// TwinCAT 3 PLC project Bangsarebuilding
// ProgramVersion: 3.1.4023.0
// libraries:
//   Tc2_EnOcean, * (Beckhoff Automation GmbH)
//   Tc2_Standard, * (Beckhoff Automation GmbH)
//   Tc2_System, * (Beckhoff Automation GmbH)
//   Tc2_Utilities, * (Beckhoff Automation GmbH)
//   Tc3_IotBase, * (Beckhoff Automation GmbH)
//   Tc3_Module, * (Beckhoff Automation GmbH)
// project tree:
//   %40Main/ MAIN.TcPOU (not stored)
//   DUTs/ ST_FrameData.TcDUT
//   / GlobalTextList.TcGTLO, PlcTask.TcTTO, Visualization Manager.TcVMO (not stored)
//   GVLs/ GVLKL3403.TcGVL, GVLmqtt.TcGVL, GVL_Enocean.TcGVL, GVL_HouseControl.TcGVL, GVL_IO_Enocean.TcGVL, GVL_RTClock.TcGVL
//   POUs/AverageLog/ FB_LoggAverage.TcPOU, NewAverage.TcPOU
//   POUs/CurrentMeassuring/ CurrentMeassuring.TcPOU, KL3403_FB.TcPOU
//   POUs/DataExchange/ DataExchange.TcPOU, F_Checksum.TcPOU
//   POUs/Enocean/ Control.TcPOU, Enocean_program.TcPOU
//   POUs/HouseControlProgram/ HouseControl.TcPOU
//   POUs/MQTT/ FB_MyMqtt.TcPOU, PrgMqttCom.TcPOU
//   POUs/RTClock/ RTClock.TcPOU
//   VISUs/VisuEnocean/ TC_VISU.TcVIS
// real-time tasks:
//   TASK PlcTask: cycle T#10ms, priority 20, ADS port 350
// I/O:
//   DEVICE Device 1 (CX-BK)
//     Box 1 (CX-BK)
// variable links:
//   Bangsarebuilding/Bangsarebuilding Instance <-> Device 1 (CX-BK)/Box 1 (CX-BK)
//     PlcTask Inputs/.DATAIN/nData <-> Term 10 (KL6021-0023)/Channel 1/Data In 0
//     PlcTask Inputs/.DATAIN/nData @bit 8 <-> Term 10 (KL6021-0023)/Channel 1/Data In 1
//     PlcTask Inputs/.DATAIN/nData @bit 80 <-> Term 10 (KL6021-0023)/Channel 1/Data In 10
//     PlcTask Inputs/.DATAIN/nData @bit 16 <-> Term 10 (KL6021-0023)/Channel 1/Data In 2
//     PlcTask Inputs/.DATAIN/nData @bit 24 <-> Term 10 (KL6021-0023)/Channel 1/Data In 3
//     PlcTask Inputs/.DATAIN/nData @bit 32 <-> Term 10 (KL6021-0023)/Channel 1/Data In 4
//     PlcTask Inputs/.DATAIN/nData @bit 40 <-> Term 10 (KL6021-0023)/Channel 1/Data In 5
//     PlcTask Inputs/.DATAIN/nData @bit 48 <-> Term 10 (KL6021-0023)/Channel 1/Data In 6
//     PlcTask Inputs/.DATAIN/nData @bit 56 <-> Term 10 (KL6021-0023)/Channel 1/Data In 7
//     PlcTask Inputs/.DATAIN/nData @bit 64 <-> Term 10 (KL6021-0023)/Channel 1/Data In 8
//     PlcTask Inputs/.DATAIN/nData @bit 72 <-> Term 10 (KL6021-0023)/Channel 1/Data In 9
//     PlcTask Inputs/.DATAIN/nStatus <-> Term 10 (KL6021-0023)/Channel 1/nStatus
//     PlcTask Inputs/.KL3403_DataIn_3 <-> Term 14 (KL3403)/Channel 1/.KL3403_DataIn_3
//     PlcTask Inputs/.KL3403_State_1 <-> Term 14 (KL3403)/Channel 1/.KL3403_State_1
//     PlcTask Inputs/.PT100_BathRoom <-> Term 13 (KL3204)/Channel 2/.PT100_BathRoom
//     PlcTask Inputs/.PT100_CX1000 <-> Term 13 (KL3204)/Channel 3/.PT100_CX1000
//     PlcTask Inputs/.PT100_Outside <-> Term 13 (KL3204)/Channel 1/.PT100_Outside
//     PlcTask Inputs/.Term3204_4_Data_In <-> Term 13 (KL3204)/Channel 4/.Term3204_4_Data_In
//     PlcTask Outputs/.AeLight <-> Term 7 (KL2012)/Channel 2/.AeLight
//     PlcTask Outputs/.AirBedroom <-> Term 3 (KL2641)/Channel 1/.AirBedroom
//     PlcTask Outputs/.AirBjorn <-> Term 2 (KL2641)/Channel 1/.AirBjorn
//     PlcTask Outputs/.BedRoomLight <-> Term 6 (KL2012)/Channel 1/.BedRoomLight
//     PlcTask Outputs/.BjornLight <-> Term 9 (KL2012)/Channel 1/.BjornLight
//     PlcTask Outputs/.DATAOUT/nCtrl <-> Term 10 (KL6021-0023)/Channel 1/nCtrl
//     PlcTask Outputs/.EntranceLight <-> Term 5 (KL2012)/Channel 2/.EntranceLight
//     PlcTask Outputs/.KL3403_Ctrl_1 <-> Term 14 (KL3403)/Channel 1/.KL3403_Ctrl_1
//     PlcTask Outputs/.KL3403_DataOut_3 <-> Term 14 (KL3403)/Channel 1/Data Out
//     PlcTask Outputs/.Livingroom <-> Term 6 (KL2012)/Channel 2/.Livingroom
//     PlcTask Outputs/.ReceptionLight <-> Term 5 (KL2012)/Channel 1/Output
//     PlcTask Outputs/.Spare <-> Term 8 (KL2012)/Channel 1/.Spare
//     PlcTask Outputs/.StairLight <-> Term 9 (KL2012)/Channel 2/.StairLight
//     PlcTask Outputs/.ToiletLight <-> Term 8 (KL2012)/Channel 2/.ToiletLight
//     PlcTask Outputs/.WalkingClosett <-> Term 7 (KL2012)/Channel 1/.WalkingClosett

CONFIGURATION Bangsarebuilding
    RESOURCE PLC ON TwinCAT3
        TASK PlcTask(INTERVAL := T#10ms, PRIORITY := 20);
        PROGRAM MAIN WITH PlcTask : MAIN;
    END_RESOURCE
END_CONFIGURATION

// ---- DUTs/ST_FrameData.TcDUT
(* 8 byte aligned structure, byte size := 152 byte *)
TYPE ST_FrameData :
STRUCT
    nFrameSize: DWORD;(*Frame byte size, member byte size := 4 byte*)
    nTxFrames : DWORD;(*Tx frame number, member byte size := 4 byte*)
    nRxFrames : DWORD;(*Rx frame number, member byte size := 4 byte*)
    nCounter  : DWORD;(*Number value, member byte size := 4 byte*)
    fU        : REAL;(*Floating point number, member byte size := 4 byte*)
    fV        : REAL;(*Floating point number, member byte size := 4 byte*)
    fW        : REAL;(*Floating point number, member byte size := 4 byte*)
    aFloats   : ARRAY[0..9] OF REAL;(* Array of floating point numbers, array byte size := 40 byte*)
    sMsg      : STRING;(*String variable, member byte size := 81 byte incl. String null delimiter*)
    bEnable   : BOOL;(*Boolean flag, member byte size := 1 byte*)
    nRsv0     : BYTE;(*Reserved byte to meet the 8 byte alignment, member byte size := 1 byte*)
    nCRC      : BYTE;(*CRC checksum byte, member byte size := 1 byte*)
END_STRUCT
END_TYPE

// ---- GVLs/GVLKL3403.TcGVL
{attribute 'Tc2GvlVarNames'}
VAR_GLOBAL
	KL3403_Ctrl_1 		AT %Q*: USINT;
	KL3403_State_1		AT %I* 	:USINT;
	KL3403_DataOut_1	 AT %Q*: INT;
	KL3403_DataIn_1	 	AT %I*	: INT;
	KL3403_Ctrl_2 		AT %Q*	: USINT;
	KL3403_State_2		AT %I* 	:USINT;
	KL3403_DataOut_2	 AT %Q*	: INT;
	KL3403_DataIn_2 		AT %I*	: INT;
	KL3403_Ctrl_3 		AT %Q*	: USINT;
	KL3403_State_3		AT %I* 	:USINT;
	KL3403_DataOut_3	 AT %Q*	: INT;
	KL3403_DataIn_3 		AT %I*	: INT;

	intOutputStatus: INT;
END_VAR

// ---- GVLs/GVLmqtt.TcGVL
{attribute 'qualified_only'}
VAR_GLOBAL

END_VAR

// ---- GVLs/GVL_Enocean.TcGVL
{attribute 'Tc2GvlVarNames'}
VAR_GLOBAL
	SummaryWordForBoolenM6 : WORD;
	OutsideTemp		: INT; 
	STM1556 :INT;

	BjornTemp 			: INT;
	OfficeTemp		 	: INT;
	BedRoomTemp 		: INT;
(* Check if enocean varible has hanged*)
	EnableForAllPTM100: BOOL := TRUE;
	CheckIfEnoceanSwitchIsPressed: DWORD;
	SRW01State: BOOL;
(*Viewer Variables*)
	EnOceanEasyClick  : BYTE; (* Status bSwitches in EnOceanEasyClick*)
	EnOceanPTM100SWbjorn :BYTE;(* Status bSwitches in EnOceanPTM100SW*)
	EnOceanPTM100SWentrance : BYTE;(* Status bSwitches in EnOceanPTM100SWentrance*)

	SRO4PeEnOceanRotarySwitch: E_EnOceanRotarySwitch;
	SRO4Psetpoint: INT;
	SRO4bPresentSwitch: BOOL;
	SRO4PbLearnSwitch: BOOL;

	SRO4P_2eEnOceanRotarySwitch: E_EnOceanRotarySwitch;
	SRO4P_2setpoint: INT;
	SRO4_2bPresentSwitch: BOOL;
	SRO4_2PbLearnSwitch: BOOL;

	SRO4P_3eEnOceanRotarySwitch: E_EnOceanRotarySwitch;
	SRO4P_3setpoint: INT;
	SRO4_3bPresentSwitch: BOOL;
	SRO4P_3bLearnSwitch: BOOL;

	SRO4PeEnOceanRotarySwitch4: E_EnOceanRotarySwitch;
	SRO4Psetpoint4: INT;
	SRO4bPresentSwitch4: BOOL;
	SRO4PbLearnSwitch4: BOOL;

(*Timers*)
	TurnLightsOffTimer: TON;
	ShutAllOff: TON;


(* Variables*)

	bLearnSTM250: BOOL;
	EnoceanResieved: ST_EnOceanReceivedData;
	EnOceanPTM100SSpareAndToilet: BYTE;
	SPir360data: ARRAY [0..3] OF BYTE;


	SRO4b3PresentSwitch: BOOL;
	SRO4P3bLearnSwitch: BOOL;
	ShutAllOff_ElapsedTime: STRING(80);
	
//	PlaceHolder_IfLightsAreON		AT %QX13.7	: BOOL;		


//	Control_ifLightsAreON 			AT %QW12: WORD;
(*	OutputControl_ifLightsAreON 				AT %QW128: WORD; (Summary word for Boolean below
	InputControl_ifLightsAreON					AT %IW132: WORD; (Summary word for Boolean below *)
END_VAR

// ---- GVLs/GVL_HouseControl.TcGVL
{attribute 'qualified_only'}
VAR_GLOBAL
//ShutAllOff(); //Maybee for later use
//ShutAllOff_ElapsedTime :=DELETE( LEFT(TIME_TO_STRING(ShutAllOff.PT-ShutAllOff.ET),5),3,0);
END_VAR

// ---- GVLs/GVL_IO_Enocean.TcGVL
{attribute 'Tc2GvlVarNames'}
VAR_GLOBAL
	DATAIN 		AT %I*: ST_EnOceanInData;
	DATAOUT 	AT %Q*: ST_EnOceanOutData;
	SpotLight		AT %Q*:	BOOL;
	ReceptionLight	AT %Q*:	BOOL;
	EntranceLight	AT %Q*:	BOOL;
	BedRoomLight	AT %Q*:	BOOL;
	Livingroom		AT %Q*:	BOOL;
	WalkingClosett	AT %Q*:	BOOL;
	AeLight			AT %Q*:	BOOL;
	BjornLight		AT %Q*:	BOOL;
	StairLight		AT %Q*:	BOOL;
	ToiletLight		AT %Q*:	BOOL;
	Spare			AT %Q*:	BOOL;
	AirBjorn 		AT %Q*: BOOL ;		
	AirBedroom 		AT %Q*: BOOL;
	TotalCurrent :	 	 INT;
	PT100_Outside		AT %I*: INT;
//	Term3403_Ctrl_1		AT %Q*: USINT;
//	Term3403_DataOut_1	AT %Q*: INT;
	PT100_BathRoom 		AT %I*: INT;
//	Term3403_Ctrl_2 		AT %Q*: USINT;
//	Term3403_DataOut_2	AT %Q*: INT;
	PT100_CX1000 		AT %I*: INT;
//	Term3403_Ctrl_3 		AT %Q*: USINT;
//	Term3403_DataOut_3	AT %Q*: INT;
//	Term3204_1_State		AT %I*:	USINT;
//	Term3204_1_Data_In	AT %I*:	INT; (*Outside*)
//	Term3204_1_Ctrl		AT %Q*:	USINT;
//	Term3204_1_Data_Out	AT %Q*:	INT;
//	Term3204_2_State		AT %IB4:USINT;
//	Term3204_2_Data_In	AT %I*:	INT;
//	Term3204_2_Ctrl		AT %Q*:	USINT;
//	Term3204_2_Data_Out	AT %Q*:	INT;
//	Term3204_3_State		AT %I*:	USINT;
//	Term3204_3_Data_In	AT %I*:	INT;
//	Term3204_3_Ctrl		AT %Q*:	USINT;
//	Term3204_3_Data_Out	AT %Q*:	INT;
//	Term3204_4_State		AT %I*:	USINT;
	Term3204_4_Data_In	AT %I*:	INT;
//	Term3204_4_Ctrl		AT %Q*:	USINT;
//	Term3204_4_Data_Out	AT %Q*:	INT;
END_VAR

// ---- GVLs/GVL_RTClock.TcGVL
{attribute 'Tc2GvlVarNames'}
VAR_GLOBAL
	stTime: TIMESTRUCT;
	PCTime: STRING;
	bRTCValid: BOOL;
	bOldWeekend: BOOL;
	OldWorkinghour: BOOL;
	OldDay: DWORD;
	OldHour: DWORD;
	OldMinute: DWORD;
//	OldSecond: DWORD;
	OldMounth: WORD;
	ChangeOfMounth: BOOL;
(*Change Variabler togels if Var has changed*)
	ChangeWeekend: BOOL;
	ChangeOfweek :BOOL;
	ChangeWorkingHour: BOOL;
	ChangeOfDay: BOOL;
	bHourChanged: BOOL;
	bMinuteChanged : BOOL;
//	bSecondCanged: BOOL;
(* Detect status*)
	bWeekend: BOOL;
	WorkingHour: BOOL;
	OldYear: WORD;
END_VAR

// ---- POUs/AverageLog/FB_LoggAverage.TcPOU
FUNCTION_BLOCK FB_LoggAverage
VAR_INPUT
	usTimeBase: USINT;(* In time i.e 60  for seconds and minutes or 24 for Hour *)
	wTIMSTR : WORD;
	rLoggdata : LREAL;
END_VAR
VAR_OUTPUT
	rAverage :LREAL ;
	arrIntern: ARRAY[0..59] OF LREAL;
END_VAR
VAR
	i: USINT;
	rMinuteAverage:  LREAL;
	//y: INT := 100;
	//: BOOL;
	//bTest: BOOL;
	usZero: USINT;
	bTimeChanged: BOOL;
	OldTimestring: WORD;	
	//arrIntern: ARRAY[0..59] OF LREAL;
END_VAR

//VAR_INPUT //old ver
//	usTimeBase: USINT;(* In time i.e 60  for seconds and minutes or 24 for Hour *)
//	wTIMSTR : WORD;
//	rLoggdata : LREAL;
//END_VAR
//VAR_OUTPUT
//	rAverage :LREAL ;
//	arrIntern : ARRAY[0..59] OF LREAL;
//END_VAR
//VAR
//	i: USINT;
//	rMinuteAverage:  LREAL;
//	y: INT := 100;
//	bFillArr: BOOL;
//	bTest: BOOL;
//	usZero: USINT;
//	bTimeChanged: BOOL;
//END_VAR

IF wTIMSTR = OldTimestring THEN
;
ELSE
bTimeChanged:= TRUE;
END_IF
OldTimestring:=wTIMSTR;
IF bTimeChanged THEN
rMinuteAverage :=0;
 arrIntern[wTIMSTR] := rLoggdata;
	IF wTIMSTR= usTimeBase -1   THEN
	usZero := usTimeBase;
		FOR i := 0 TO usTimeBase -1  DO
			IF arrIntern[i] = 0 THEN
			usZero := usZero - 1;
			END_IF
		rMinuteAverage := arrIntern[i]+ rMinuteAverage;
arrIntern[i] := 0;

 			IF i = usTimeBase -1 THEN
				IF usZero = 0 THEN
				RETURN ;
				END_IF
	 		rAverage := rMinuteAverage / (usZero ) ;
			bTimeChanged := FALSE ;
			END_IF
		END_FOR
	END_IF
END_IF

END_FUNCTION_BLOCK

// ---- POUs/AverageLog/NewAverage.TcPOU
PROGRAM NewAverage
VAR
	rAverageMin: LREAL;
	rAverageHour: LREAL;
	rAverageDay : LREAL;
	rLoggData: LREAL ;
	FB_LoggAverageMonth: FB_LoggAverage;
	FB_LoggAverageDays:  FB_LoggAverage;
	FB_LoggAverageHours: FB_LoggAverage;
	FB_LoggAverageMinutes: FB_LoggAverage;
	FB_LoggAverageSeconds: FB_LoggAverage;
(*	arrZeros : ARRAY[0..9 ]  OF sDataLogg; *)

	rTestData: REAL;
	rAverageMonth: LREAL;
	rAverageYear: LREAL;
END_VAR


rLoggData := .TotalCurrent; //Test
FB_LoggAverageSeconds(
	usTimeBase:=60 ,
	wTIMSTR := GVL_RTClock.stTime.wSecond, (* Array index *)
	rLoggData:= rLoggData ,							(**)
	rAverage=> rAverageMin);

FB_LoggAverageMinutes(
	usTimeBase:=60 ,
	wTIMSTR := GVL_RTClock.stTIME. wMinute, (* Array index *)
	rLoggData:= rAverageMin ,							(**)
	rAverage=> rAverageHour );

FB_LoggAverageHours(
	usTimeBase:=24 ,
	wTIMSTR := GVL_RTClock.stTIME. wHour  , (* Array index *)
	rLoggData:= rAverageHour ,
	rAverage=> rAverageDay) ;

FB_LoggAverageDays( 
	usTimeBase:= 31,
	wTIMSTR := GVL_RTClock.stTime.wDay, (* Array index *)
	rLoggData:= rAverageDay ,
	rAverage =>rAverageMonth);

FB_LoggAverageMonth( 
	usTimeBase:= 31,
	wTIMSTR := GVL_RTClock.stTime.wMonth, (* Array index *)
	rLoggData:= rAverageMonth ,
	rAverage =>rAverageYear);

END_PROGRAM

// ---- POUs/CurrentMeassuring/CurrentMeassuring.TcPOU
PROGRAM CurrentMeassuring
VAR
	bEnable: BOOL := TRUE;
	arrPowerMeasure1: ARRAY [0..11] OF INT;
	arrPowerMeasure2 : ARRAY [0..11] OF INT;
	arrPowerMeasure3 : ARRAY [0..11] OF INT;
	fb_Ch1: KL3403_FB;
(*	fb_Ch2: KL3403_FB;
	fb_Ch3: KL3403_FB;*)
	intOldHour: INT;
	arrLoggHour: ARRAY [0..1,0..23] OF REAL;
	intOldDay: INT;
	arrDataYesterday: ARRAY [0..1,0..23] OF REAL;
	realCurrentRMS: REAL;
	realVoltageRMS: REAL;
	realEff_Power: REAL;
	realPF: REAL;
	realPeakCurrent: REAL;
	realPeakVoltage: REAL;
	realPeakPower: REAL;
	realHz: REAL;
	realMinCurrent: REAL;
	realMinVoltage: REAL;
END_VAR
VAR_INPUT
	intState: USINT;
END_VAR

(*
fb_Ch1(
	bEnable:= TRUE,
	usintState:= KL3403_State_1,
	intDataIN:=KL3403_DataIn_1 ,
	usintCTRL=>KL3403_Ctrl_1 ,
	arrPowerMeasure => arrPowerMeasure1,
	realCurrentRMS=> intCurrentLamp1,
	realVoltageRMS=>intVoltage1


fb_Ch2(
	bEnable:= TRUE,
	usintState:= KL3403_State_2,
	intDataIN:=KL3403_DataIn_2 ,
	usintCTRL=>KL3403_Ctrl_2 ,
	arrPowerMeasure => arrPowerMeasure2,
	realCurrentRMS=> intCurrentLamp2,
	realVoltageRMS=>intVoltage2
 );
 *)
fb_Ch1(
	bEnable:= TRUE,
	usintState:= KL3403_State_3,
	intDataIN:=KL3403_DataIn_3 ,
	usintCTRL=>KL3403_Ctrl_3 ,
	arrPowerMeasure => arrPowerMeasure3,
//	realCurrentRMS=>intCurrentSolar ,
//	realVoltageRMS=>intVoltage3
 );

arrPowerMeasure1[0];
arrPowerMeasure1[1];
.TotalCurrent := KL3403_DataIn_3;

fb_Ch1(
	bEnable:= bEnable,
	usintState:= KL3403_State_3,
	intDataIN:= KL3403_DataIn_3,
	usintCTRL=>KL3403_Ctrl_3 ,
	arrPowerMeasure => arrPowerMeasure2,
	realCurrentRMS=> realCurrentRMS, 
	realVoltageRMS=>realVoltageRMS ,
	realEff_Power=>realEff_Power , 
	realPF=>realPF , 
	realEnergyConsumtion=> , 
	realPeakCurrent=>realPeakCurrent ,
	realPeakVoltage=> realPeakVoltage,
	realPeakPower=> realPeakPower, 
	realHz=>realHz , 
	realMinCurrent=> realMinCurrent, 
	realMinVoltage=> realMinVoltage, 
	realMinPower=> realMinVoltage );

END_PROGRAM

// ---- POUs/CurrentMeassuring/KL3403_FB.TcPOU
FUNCTION_BLOCK KL3403_FB
VAR
	TP1: TP;
	TP2: TP;
	R_TRIG1: R_TRIG;

	INDEX: BYTE;
	CurrentRMS: REAL;
	VoltageRMS: REAL;
	EffectivePower: REAL;
	PowerFactor: REAL;
	EnergyConsuntion: REAL;
	PeakCurrent: REAL;
	PeakVoltage: REAL;
	PeakPower: REAL;
	Frequency: REAL;
	MinimumCurrent: REAL;
	MinimumVoltage: REAL;
	MinimumPower: REAL;
END_VAR
VAR_INPUT
	bEnable: BOOL;
	usintState : INT;
	intDataIN: INT;
END_VAR
VAR_OUTPUT
	usintCTRL: USINT;
	arrPowerMeasure: ARRAY [0..11] OF INT;
	realCurrentRMS: REAL;
	realVoltageRMS: REAL;
	realEff_Power: REAL;
	realPF: REAL;
	realEnergyConsumtion: REAL;
	realPeakCurrent: REAL;
	realPeakVoltage: REAL;
	realPeakPower: REAL;
	realHz: REAL;
	realMinCurrent: REAL;
	realMinVoltage: REAL;
	realMinPower: REAL;
END_VAR

(* Update Value form KL3403*)

usintCTRL := index ;
IF usintState.0 = usintCTRL.0 THEN
arrPowerMeasure[index] := intDataIN ;
index := index +1;
END_IF
IF index >11 THEN Index := 0 ; END_IF

(*Transfer data*)


(*Show in Function Block Output*)
realCurrentRMS :=INT_TO_REAL (arrPowerMeasure[0]);
realVoltageRMS := INT_TO_REAL (arrPowerMeasure[1])/10.0;
realEff_Power := INT_TO_REAL( arrPowerMeasure[2]);
realPF := INT_TO_REAL (arrPowerMeasure[3] ) ;
realEnergyConsumtion := INT_TO_REAL (arrPowerMeasure[4] ) ;
realPeakCurrent := INT_TO_REAL (arrPowerMeasure[4]) ;
realPeakVoltage := INT_TO_REAL (arrPowerMeasure[4])/10.0;
realPeakPower := INT_TO_REAL (arrPowerMeasure[4]) ;
realHz :=INT_TO_REAL (arrPowerMeasure[4])/10.0;
realMinCurrent := INT_TO_REAL( arrPowerMeasure[4]);
realMinVoltage := INT_TO_REAL (arrPowerMeasure[4] )/ 10.0;
realMinPower := INT_TO_REAL (arrPowerMeasure[4]);

END_FUNCTION_BLOCK

// ---- POUs/DataExchange/DataExchange.TcPOU
PROGRAM DataExchange
VAR
    bWrite        : BOOL;(* Rising edge at this variable writes data to the BC/BX (Bus Terminal Controller) *)
    bRead         : BOOL;(* Rising edge at this variable reads data from BC/BX (Bus Terminal Controller) *)
    stTxFrame     : ST_FrameData; (* Data transported from PC/CX (x86) to BC/BX (Bus Terminal Contoroller) *)
    stRxFrame     : ST_FrameData; (* Data transported from BC/BX (Bus Terminal Controller) to PC/CX (x86) *)
    fbWrite       : ADSWRITE :=  ( NETID := '172.16.5.128.1.1', PORT := 800, IDXGRP := 16#4020, IDXOFFS := 500, TMOUT := DEFAULT_ADS_TIMEOUT );
    fbRead        : ADSREAD :=  ( NETID := '172.16.5.128.1.1', PORT := 800, IDXGRP := 16#4020, IDXOFFS := 0, TMOUT := DEFAULT_ADS_TIMEOUT );
    (* Temporary used variables *)
    stTxToBC      : ST_FrameData;
    stRxFromBC    : ST_FrameData;
    i             : INT;
    nTxState      : UDINT;
    nRxState      : UDINT;
    nTxErrors     : UDINT;
    nRxErrors     : UDINT;
END_VAR

(*##########################################################################################*)
CASE nTxState OF
    0:
        IF bWrite THEN(* Write BC/BX data *)
            bWrite := FALSE;

            (* Prepare/modify tx data *)
            stTxFrame.nFrameSize    := SIZEOF( stTxFrame );(* Set frame byte size *)
            stTxFrame.nTxFrames    := stTxFrame.nTxFrames + 1;(* Increment the send frame number *)
            stTxFrame.nRxFrames     := stRxFrame.nTxFrames;(* Report the received frame number *)
            stTxFrame.bEnable    := NOT stTxFrame.bEnable;(* Toggle bool flag *)
            stTxFrame.nCounter     := stTxFrame.nCounter + 1;(* Increment counter value *)
            stTxFrame.sMsg         := CONCAT( 'Message from PC/CX, counter: ', DWORD_TO_STRING( stTxFrame.nCounter ) );(* Create some string message *)
            stTxFrame.fU            := stTxFrame.fU + 1.2;(* Modify some floating point values *)
            stTxFrame.fV            := stTxFrame.fV + 3.4;
            stTxFrame.fW            := stTxFrame.fW + 5.6;
            FOR i:= 0 TO 9 DO
                stTxFrame.aFloats[i] := stTxFrame.aFloats[i] + i;
            END_FOR
            stTxFrame.nCRC         := 0;

            (* Create temporary copy of tx data *)
            stTxToBC := stTxFrame;

            (* Swap REAL variables to BC/BX (Bus Terminal Controller) format *)
            F_SwapRealEx( stTxToBC .fU );
            F_SwapRealEx( stTxToBC .fV );
            F_SwapRealEx( stTxToBC .fW );
            FOR i:= 0 TO 9 DO
                F_SwapRealEx( stTxToBC .aFloats[i] );
            END_FOR
    
            (* Create CRC check number *)
            stTxToBC .nCRC     := F_CheckSum( ADR( stTxToBC ), SIZEOF( stTxToBC ) - 1 );
    
            (* Send *)
            fbWrite( WRITE := FALSE );
            fbWrite( LEN := SIZEOF( stTxToBC ), SRCADDR := ADR( stTxToBC ), WRITE := TRUE );
            nTxState := 1;
        END_IF

    1:(* Wait until ads write command not busy *)
        fbWrite( WRITE := FALSE );
        IF NOT fbWrite.BUSY THEN
            IF NOT fbWrite.ERR THEN
                nTxState := 0;
            ELSE(* Ads error *)
                nTxState := 100;
            END_IF
        END_IF

    100: (* TODO: Error state, add error handling *)
        nTxErrors := nTxErrors + 1;
        nTxState := 0;

END_CASE

(*##########################################################################################*)
CASE nRxState OF
    0:
        IF bRead THEN(* Read BC/BX data *)
            bRead := FALSE;

            fbRead( READ := FALSE );
            fbRead( LEN := SIZEOF( stRxFromBC ), DESTADDR := ADR( stRxFromBC ), READ := TRUE );
            nRxState := 1;
        END_IF

    1:(* Wait until ads read command not busy *)
        fbRead( READ := FALSE );
        IF NOT fbRead.BUSY THEN
            IF NOT fbRead.ERR THEN
                (* Perform simple frame length check *)
                IF stRxFromBC.nFrameSize = SIZEOF( stRxFromBC ) THEN (* Check frame length *)
                    (* Perform simple CRC check *)
                    IF stRxFromBC.nCRC = F_CheckSum( ADR( stRxFromBC ), SIZEOF( stRxFromBC ) - 1 ) THEN

                        (* Swap REAL variables to PC/CX (x86) format *)
                        F_SwapRealEx( stRxFromBC.fU );
                        F_SwapRealEx( stRxFromBC.fV );
                        F_SwapRealEx( stRxFromBC.fW );
                        FOR i:= 0 TO 9 DO
                            F_SwapRealEx( stRxFromBC.aFloats[i] );
                        END_FOR

                        stRxFrame := stRxFromBC;
                        nRxState     := 0;

                    ELSE(* => Checksum error *)
                        nRxState := 100;
                    END_IF
                ELSE(* => Invalid frame length *)
                    nRxState := 100;
                END_IF
            ELSE(* => Ads error *)
                nRxState := 100;
            END_IF
        END_IF

    100: (* TODO: Error state, add error handling *)
        nRxErrors := nRxErrors + 1;
        nRxState := 0;

END_CASE

END_PROGRAM

// ---- POUs/DataExchange/F_Checksum.TcPOU
FUNCTION F_Checksum : BYTE
VAR_INPUT
	pBuffer 		: POINTER TO BYTE;
	cbBuffer 	: UDINT;
END_VAR
VAR
	i			: UDINT;
END_VAR

IF ( pBuffer = 0 ) OR ( cbBuffer = 0 ) THEN
	F_CheckSum := 0;
	RETURN;
END_IF

FOR i:= 1 TO cbBuffer DO
	F_CheckSum := F_CheckSum + pBuffer^;
	pBuffer := pBuffer + 1;
END_FOR

END_FUNCTION

// ---- POUs/Enocean/Control.TcPOU
PROGRAM Control
VAR
	rtrigStairs: R_TRIG;
	rtrigBjorn: R_TRIG;
	rtrigBalcony: R_TRIG;
	rtrigWindow: R_TRIG;
	rtrigToilet: R_TRIG;
	rtrigBedroom: R_TRIG;
	rtrigEntrance: R_TRIG;
	rtrigSofa: R_TRIG;
	rtrigSpotlight: R_TRIG;
	rtrigReception: R_TRIG;
	rtrigEntrance2: R_TRIG;
	rtrigSofa2: R_TRIG;
	rtrigSpotlight2: R_TRIG;
	rtrigReception2: R_TRIG;
	rtrigPreparationToLeave: R_TRIG;
	Delay: TIME := T#10S;
	OffTimerPTM100SWbjorn: TON;
	OffTimerPTM100SWentrance:TON;
	OffTimerEasyClick:TON;
	OffTimerSpareAndToilet: TON;
	OldSummaryWordForBoolenM6: WORD;
	VBchange: BOOL;
	TON_InputHanged: TON;
	TimerFoorAirBedroom: TON;
	WorkingHourTest: BOOL;
	rtrig4: R_TRIG;
	rtrig5: R_TRIG;
	rtrig1: R_TRIG;
	rtrig0: R_TRIG;
	A: UINT;
	bTest: BOOL;
END_VAR



Control.EasyfitBjorn();(* Action uses data from Switch at Room Bjorn*)
Control.EasyFitSpareAndToiletUppstairs();(* Action uses data from Switch at Spareroom and Toilet uppstairs*)
Control.EasyfitEntrance(); (* Action uses data from Switch at entrance door*)

ACTION EasyfitBjorn:
(* EasyfitBjornEasyfitEntrance has 4 buttons, controling 4 lamps press a button is on and if same button is prssed more than 1sec light goes off
Data is evalueted in MAIN.EntrancewitchControl.EnOceanPTM100SWbjorn, i.e. .bSw0 to bSw3 are set when corresponding switch is pressed *)

rtrigStairs(CLK:=Enocean_program.fb_PTM100SWbjorn1159899.bSwitches[4] );
rtrigBjorn(CLK := Enocean_program.fb_PTM100SWbjorn1159899.bSwitches[5]);
rtrigBalcony(CLK := Enocean_program.fb_PTM100SWbjorn1159899.bSwitches[1]);
rtrigWindow(CLK := Enocean_program.fb_PTM100SWbjorn1159899.bSwitches[0]);

IF rtrigStairs.Q THEN
StairLight := NOT StairLight;
END_IF
IF rtrigBalcony.Q THEN
	Livingroom:= NOT Livingroom ;
END_IF
IF rtrigBjorn.Q THEN
	BjornLight :=NOT BjornLight;
END_IF
IF rtrigWindow.Q THEN
	BedRoomLight := NOT BedRoomLight;
END_IF
END_ACTION

ACTION EasyfitEntrance:
(* EasyfitEntrance has 4 buttons, controling 4 lamps. 2 Switches doing the same jobb are used *)

rtrigEntrance(CLK:= Enocean_program.fb_PTM100SWentrance1119127.bSwitches[5]  );
rtrigSofa(CLK:=  Enocean_program.fb_PTM100SWentrance1119127.bSwitches[1] );
rtrigSpotlight(CLK:= Enocean_program.fb_PTM100SWentrance1119127.bSwitches[4]   );
rtrigReception(CLK:= Enocean_program.fb_PTM100SWentrance1119127.bSwitches[0]  );
(*
rtrigEntrance2(CLK:= Enocean_program.fb_PTM100SWentrance1119127.bSwitches[5]  );
rtrigSofa2(CLK:=  Enocean_program.fb_PTM100SWentrance1119127.bSwitches[1] );
rtrigSpotligh2t(CLK:= Enocean_program.fb_PTM100SWentrance1119127.bSwitches[4]   );
rtrigReception2(CLK:= Enocean_program.fb_PTM100SWentrance1119127.bSwitches[0]  );
*)


(*Turn On and Off  Light at Entrance*)

IF rtrigEntrance.Q  THEN(* Upper left switch *)
	ReceptionLight := NOT ReceptionLight;
END_IF
IF rtrigSofa.Q  THEN(*Lower Left SW*)
	AeLight := NOT AeLight;
	(*IF NOT DayTime THEN	Stairs :=TRUE; END_IF*)
END_IF

IF rtrigSpotlight.Q THEN (* Upper right switch *)
	SpotLight := NOT SpotLight;
END_IF
IF rtrigReception.Q THEN(*Lower Left SW*)
	ReceptionLight := NOT ReceptionLight;
END_IF

(*
IF rtrigEntrance2.Q  THEN(* Upper left switch *)
	Entrance := NOT Entrance;
END_IF
IF rtrigSofa2.Q  THEN(*Lower Left SW*)
	Sofa := NOT Sofa;
	IF NOT WorkingHour THEN	Stairs :=TRUE; END_IF
END_IF

IF rtrigSpotlight2.Q THEN (* Upper right switch *)
	Spotlight := NOT Spotlight;
END_IF
IF rtrigReception2.Q THEN(*Lower Left SW*)
	Reception := NOT Reception;
END_IF
*)
END_ACTION

ACTION EasyFitSpareAndToiletUppstairs:
(* EasyFitSpareAndToiletUppstairs has 2buttons, controling 2 lamps press a button is on and if same button is prssed more than 1sec light goes off
Data is evalueted in MAIN.EntrancewitchControl.EasyFitSpareAndToiletUppstairs, i.e. .bSw0 to bSw3 are set when corresponding switch is pressed *)
rtrigToilet (CLK:= Enocean_program.fb_PTM100SWSpareAndToilet1075788.bSwitches[5] , Q=> );
rtrigBedroom(CLK:= Enocean_program.fb_PTM100SWSpareAndToilet1075788.bSwitches[1]  , Q=> );
IF rtrigToilet.Q  THEN
	ToiletLight:=NOT ToiletLight;
END_IF
IF rtrigBedroom.Q THEN
	BedRoomLight := NOT  BedRoomLight;
END_IF
END_ACTION

END_PROGRAM

// ---- POUs/Enocean/Enocean_program.TcPOU
PROGRAM Enocean_program (* Evaluates in _RECIVER if an Enocean signal is activated
							the other fb:s controls variables  depending on Enoceandata recieved.*)
VAR_INPUT
END_VAR
VAR
	FB_EnOceanReceive1: FB_EnOceanReceive;
	fb_BeckhoffSooftSW4294378625	:FB_EnOceanPTM100;
	fb_PTM100SWentrance1119127		: FB_EnOceanPTM100;
	fb_PTM100SWbjorn1159899			: FB_EnOceanPTM100;
	fb_PTM100SWSpareAndToilet1075788: FB_EnOceanPTM100;
	FB_EnOceanSTM100				: FB_EnOceanSTM100;
	FB_EnOceanSTM1556				: FB_EnOceanSTM100;
	FB_EnOceanSTM100_2				: FB_EnOceanSTM100;
	FB_EnOceanSTM100_3				: FB_EnOceanSTM100;
	FB_EnOceanSTM100_4				: FB_EnOceanSTM100;
	FB_EnOceanSTM250				: FB_EnOceanSTM250;
	FB_EnOceanSTM100PIR360			: FB_EnOceanSTM100Generic;
	bSwitches:ARRAY[0..7] OF BOOL ;
	bError: BOOL;
	nErrorId: UDINT;
	PresentTransmiterId: UDINT;
	FB_EnOceanReceive2: FB_EnOceanReceive;
	ui1556: INT;
	ui1936: INT;
	ui58058: INT;
	ui58059: INT;
	ui58398: INT;
END_VAR

(*1138914  Evaluates in _RECIVER if an Enocean signal  is activated, the other fb:s sets a variables  depending on Enoceandata recieved.*)
FB_EnOceanReceive1(
	bEnable:= TRUE, 
	bError=> , 
	nErrorId=> , 
	stEnOceanReceivedData=> EnoceanResieved, 
	stEnOceanInData:= DATAIN , 
	stEnOceanOutData:= DATAOUT);
//FB_EnOceanReceive1				(
//								bEnable:=TRUE ,
//								stEnOceanInData:=DATAIN ,
//								stEnOceanOutData:=DATAOUT ,	
//								bError=> ,	
//								nErrorId=> ,	
//								stEnOceanReceivedData=>EnoceanResieved );
								
fb_PTM100SWentrance1119127	(bEnable:= EnableForAllPTM100,	tWatchdog:=,	nTransmitterId:=1119127 ,	stEnOceanReceivedData:= FB_EnOceanReceive1.stEnOceanReceivedData,
										bSwitches=>,	bError=> ,	nErrorId=> );
fb_PTM100SWbjorn1159899		(	bEnable:= EnableForAllPTM100,	tWatchdog:=,	nTransmitterId:= 1159899,	stEnOceanReceivedData:= FB_EnOceanReceive1.stEnOceanReceivedData,
										bSwitches=>,	bError=> ,	nErrorId=> );
fb_PTM100SWSpareAndToilet1075788(	bEnable:= EnableForAllPTM100,	tWatchdog:=,	nTransmitterId:= 1075788,	stEnOceanReceivedData:= FB_EnOceanReceive1.stEnOceanReceivedData,
										bSwitches=>,	bError=> ,	nErrorId=> );
fb_BeckhoffSooftSW4294378625 (bEnable:= EnableForAllPTM100,
							    tWatchdog:=,	nTransmitterId:= 1406393,
								stEnOceanReceivedData:= FB_EnOceanReceive1.stEnOceanReceivedData,
								bSwitches=>bSwitches,
								bError=>bError ,
								nErrorId=>nErrorId );

FB_EnOceanSTM100					(bEnable:=TRUE ,	tWatchdog:=T#30m ,	nTransmitterId:=58398 ,	stEnOceanReceivedData:=FB_EnOceanReceive1.stEnOceanReceivedData ,
										 eEnOceanRotarySwitch=>SRO4PeEnOceanRotarySwitch  ,	nSetpoint=>SRO4Psetpoint ,	nTemperature=> ,	bPresentSwitch=>SRO4bPresentSwitch ,
										bLearnSwitch=>SRO4PbLearnSwitch ,bError=> ,	nErrorId=> );
FB_EnOceanSTM1556					(bEnable:=TRUE ,	tWatchdog:=T#30M ,	nTransmitterId:=1556 ,	stEnOceanReceivedData:=FB_EnOceanReceive1.stEnOceanReceivedData ,
										 eEnOceanRotarySwitch=>SRO4PeEnOceanRotarySwitch  ,	nSetpoint=>SRO4Psetpoint ,	nTemperature=> ,	bPresentSwitch=>SRO4bPresentSwitch ,
										bLearnSwitch=>SRO4PbLearnSwitch ,bError=> ,	nErrorId=> );										
FB_EnOceanSTM100_2			(	bEnable:=TRUE ,	tWatchdog:=T#30m ,	nTransmitterId:=58058 ,	stEnOceanReceivedData:=FB_EnOceanReceive1.stEnOceanReceivedData ,
										eEnOceanRotarySwitch=>SRO4P_2eEnOceanRotarySwitch  ,	nSetpoint=>SRO4P_2setpoint ,	nTemperature=> ,	bPresentSwitch=>SRO4_2bPresentSwitch ,
										bLearnSwitch=>SRO4_2PbLearnSwitch ,	bError=> ,	nErrorId=> );
FB_EnOceanSTM100_3			(	bEnable:=TRUE ,	tWatchdog:=T#30m ,	nTransmitterId:=58059 ,	stEnOceanReceivedData:=FB_EnOceanReceive1.stEnOceanReceivedData ,
										eEnOceanRotarySwitch=>SRO4PeEnOceanRotarySwitch  ,	nSetpoint=>SRO4P_3setpoint ,	nTemperature=> ,	bPresentSwitch=>SRO4_3bPresentSwitch ,
										bLearnSwitch=>SRO4P_3bLearnSwitch ,	bError=> ,	nErrorId=> );
FB_EnOceanSTM100_4			(	bEnable:=TRUE ,	tWatchdog:=T#30m ,	nTransmitterId:=1936 ,	stEnOceanReceivedData:=FB_EnOceanReceive1.stEnOceanReceivedData ,
										eEnOceanRotarySwitch=>SRO4PeEnOceanRotarySwitch4  ,	nSetpoint=>SRO4Psetpoint4 ,	nTemperature=> ,	bPresentSwitch=>SRO4bPresentSwitch4 ,
										bLearnSwitch=>SRO4PbLearnSwitch4 ,	bError=> ,	nErrorId=> );

FB_EnOceanSTM100PIR360		(	bEnable:=TRUE ,	tWatchdog:=T#30m ,	nTransmitterId:=41490 ,	stEnOceanReceivedData:=FB_EnOceanReceive1.stEnOceanReceivedData ,
										nDataBytes=>SPir360data ,	bError=> ,	nErrorId=> );
FB_EnOceanSTM250				(	bEnable:=TRUE ,	tWatchdog:= ,	nTransmitterId:=25391 ,	stEnOceanReceivedData:=FB_EnOceanReceive1.stEnOceanReceivedData,
										bState=>SRW01State ,	bLearn=> bLearnSTM250,	bError=> , 	nErrorId=> );

(* Temperature is present in 1/10 grad i.e 312 means 31.2 grad*)
PresentTransmiterId:=EnoceanResieved.nTransmitterId;
 CASE PresentTransmiterId OF
1556: ui1556 := ui1556 + 1;	 
1936: ui1936 := ui1936 + 1;
58058: ui58058 := ui58058 + 1;
58059: ui58059 := ui58059 + 1;
58398:	ui58398 := ui58398 + 1; 
 END_CASE
OutsideTemp  :=FB_EnOceanSTM100.nTemperature;
OfficeTemp :=FB_EnOceanSTM100_2.nTemperature ;
STM1556 := FB_EnOceanSTM1556.nTemperature ;
BedRoomTemp :=FB_EnOceanSTM100_3.nTemperature ;
BjornTemp:=FB_EnOceanSTM100_4.nTemperature;


(* the array bSwitches is really 8 BYTE using only 1 bit as Boolean.
Below they are converted to bit in 1 WORD. evaluated in CheckIfHanged*) 
EnOceanEasyClick.0 :=FB_BeckhoffSooftSW4294378625.bSwitches[0];
EnOceanEasyClick.1 :=FB_BeckhoffSooftSW4294378625.bSwitches[1];
EnOceanEasyClick.4 :=FB_BeckhoffSooftSW4294378625.bSwitches[4];
EnOceanEasyClick.5 :=FB_BeckhoffSooftSW4294378625.bSwitches[5];

EnOceanPTM100SWbjorn.0 :=fb_PTM100SWbjorn1159899.bSwitches[0];
EnOceanPTM100SWbjorn.1 :=fb_PTM100SWbjorn1159899.bSwitches[1];
EnOceanPTM100SWbjorn.4 :=fb_PTM100SWbjorn1159899.bSwitches[4];
EnOceanPTM100SWbjorn.5 :=fb_PTM100SWbjorn1159899.bSwitches[5];

EnOceanPTM100SWentrance.0 :=fb_PTM100SWentrance1119127.bSwitches[0];
EnOceanPTM100SWentrance.1 :=fb_PTM100SWentrance1119127.bSwitches[1];
EnOceanPTM100SWentrance.4 :=fb_PTM100SWentrance1119127.bSwitches[4];
EnOceanPTM100SWentrance.5 :=fb_PTM100SWentrance1119127.bSwitches[5];

EnOceanPTM100SSpareAndToilet.1 :=fb_PTM100SWSpareAndToilet1075788.bSwitches[1];
EnOceanPTM100SSpareAndToilet.5 :=fb_PTM100SWSpareAndToilet1075788.bSwitches[5];

(*
Not used in PTM Switch with 2 channels
EnOceanPTM100SSpareAndToilet.0 :=fb_PTM100SWSpareAndToilet1075788.bSwitches[0];
EnOceanPTM100SSpareAndToilet.2 :=fb_PTM100SWSpareAndToilet1075788.bSwitches[2];
EnOceanPTM100SSpareAndToilet.3 :=fb_PTM100SWSpareAndToilet1075788.bSwitches[3];
EnOceanPTM100SSpareAndToilet.4 :=fb_PTM100SWSpareAndToilet1075788.bSwitches[4];
EnOceanPTM100SSpareAndToilet.6 :=fb_PTM100SWSpareAndToilet1075788.bSwitches[6];
EnOceanPTM100SSpareAndToilet.7 :=fb_PTM100SWSpareAndToilet1075788.bSwitches[7];
*)

END_PROGRAM

// ---- POUs/HouseControlProgram/HouseControl.TcPOU
PROGRAM HouseControl
VAR

END_VAR


IF stTime.wHour = 18 AND stTime.wMinute =1 THEN
StairLight := TRUE; //Cant be shut off for 1 minute 
ELSIF stTime.wHour = 23 AND stTime.wMinute =59 THEN
StairLight := TRUE; //Cant be shut off for 1 minute 	
END_IF

END_PROGRAM

// ---- POUs/MQTT/FB_MyMqtt.TcPOU
{attribute 'c++_compatible'}
FUNCTION_BLOCK FB_MyMqtt EXTENDS FB_IotMqttClient
VAR_INPUT
END_VAR
VAR_OUTPUT
END_VAR

VAR
	(* received message *)
	{attribute 'TcEncoding':='UTF-8'}
	sTopicRcv : STRING(255);
	{attribute 'TcEncoding':='UTF-8'}
	sPayloadRcv : STRING(255);
	A: BOOL;
	nVar: INT;
END_VAR

{attribute 'c++_compatible'}
{attribute 'pack_mode' := '4'}
{attribute 'show'}
{attribute 'minimal_input_size' := '4'}
METHOD OnMqttMessage : HRESULT
VAR_IN_OUT CONSTANT
	topic	: STRING;
END_VAR
VAR_INPUT
	payload	: PVOID;
	length	: UDINT;
	qos	: TcIotMqttQos;
	repeated	: BOOL;
END_VAR

VAR
	sRecived: STRING(255);
Test :int ;
END_VAR
SUPER^.nMessagesRcv := SUPER^.nMessagesRcv + 1;

STRNCPY( ADR(sTopicRcv), ADR(topic), SIZEOF(sTopicRcv) );
MEMCPY( ADR(sPayloadRcv), payload, MIN(length, DINT_TO_UDINT(SIZEOF(sPayloadRcv))) );
sTopicRcv;
sPayloadRcv;
nVar := STRING_TO_INT(sPayloadRcv);
IF sTopicRcv = 'BangsareLights' THEN
      CASE nVar OF 
		  0: ;
		  1:  SpotLight := NOT SpotLight;
		  2:  ReceptionLight := NOT ReceptionLight ;
		  3:  EntranceLight := NOT EntranceLight;
		  4:  BedRoomLight := NOT BedRoomLight;
		  5:  Livingroom := NOT Livingroom;
		  6:  WalkingClosett := NOT WalkingClosett;
		  7:  BjornLight := FALSE;
		  8:  BjornLight := TRUE;
		  9:  StairLight := FALSE;
		  10: StairLight := TRUE;
		  11: Spare := NOT Spare;
	  END_CASE
	  	Test :=Test +1;
	END_IF
	sPayloadRcv:='0';
OnMqttMessage := S_OK;
END_METHOD

END_FUNCTION_BLOCK

// ---- POUs/MQTT/PrgMqttCom.TcPOU
PROGRAM PrgMqttCom
VAR
	fbMqttClient : FB_MyMqtt;
	bSetParameter : BOOL := TRUE;
	bConnect : BOOL := TRUE;
	
	(* published message *)
	sTopicPub : STRING(255) := 'MyTopic';
	sPayloadPub : STRING(255);
	i: UDINT;
	fbTimer : TON := (PT:=T#1S);
	
	bSubscribed : BOOL;
	sTopicSub : STRING(255) := 'MyTopic';
	
	hrErrorOccurred : HRESULT; // contains the latest occurred error
	fbTimerET: TIME;
	bFbTimer: BOOL;
	Value: UDINT;
END_VAR

IF bSetParameter THEN
	bSetParameter := FALSE;
	fbMqttClient.sHostName:= 'SERVICE';
	fbMqttClient.nHostPort:= 1883;
	fbMqttClient.sClientId:= 'IotMqttSample'; 
	fbMqttClient.sTopicPrefix:= ''; 
//	fbMqttClient.nKeepAlive:= 60; 
//	fbMqttClient.sUserName:= ;
//	fbMqttClient.sUserPassword:= ; 
//	fbMqttClient.stTLS:= ;
 	fbMqttClient.stWill.sTopic := 'LASTWILL';
//	fbMqttClient.stWill.pPayload:= 'IotMqttSample';
	fbMqttClient.stWill.nPayloadSize := Value;
END_IF

fbMqttClient.Execute(bConnect);
IF fbMqttClient.bError THEN
	// add your error logging here
	hrErrorOccurred := fbMqttClient.hrErrorCode;
END_IF
//Add Subscribe here
IF fbMqttClient.bConnected THEN
	IF NOT bSubscribed THEN
		bSubscribed := fbMqttClient.Subscribe(sTopic:=sTopicSub, eQoS:=TcIotMqttQos.AtMostOnceDelivery);
		bSubscribed := fbMqttClient.Subscribe(sTopic:='motorCurrent', eQoS:=TcIotMqttQos.AtMostOnceDelivery);
		bSubscribed := fbMqttClient.Subscribe(sTopic:='motorTemp', eQoS:=TcIotMqttQos.AtMostOnceDelivery);
		bSubscribed := fbMqttClient.Subscribe(sTopic:='motorVoltage', eQoS:=TcIotMqttQos.AtMostOnceDelivery);
		bSubscribed := fbMqttClient.Subscribe(sTopic:='BangsareLights', eQoS:=TcIotMqttQos.AtMostOnceDelivery);
		IF fbMqttClient.bError THEN
			// add your error logging here
			hrErrorOccurred := fbMqttClient.hrErrorCode;
		END_IF
	END_IF
	//Add Publish here
	fbTimer(IN:=bFbTimer , PT:=T#10S , Q=> , ET=>fbTimerET );
	IF fbTimer.Q THEN // publish new payload every second // Changed to minute
		fbTimer(IN:=FALSE);
		i := i + 1;
		sPayloadPub := CONCAT('MyMessage', TO_STRING(i));
		fbMqttClient.Publish(	sTopic:= sTopicPub, 
								pPayload:= ADR(sPayloadPub), nPayloadSize:= LEN2(ADR(sPayloadPub))+1, 
								eQoS:= TcIotMqttQos.AtMostOnceDelivery, bRetain:= FALSE, bQueue:= FALSE );
		IF fbMqttClient.bError THEN
			// add your error logging here
			hrErrorOccurred := fbMqttClient.hrErrorCode;
		END_IF
	END_IF
END_IF

END_PROGRAM

// ---- POUs/RTClock/RTClock.TcPOU
PROGRAM RTClock
VAR
	fbGetLocalTime  	: NT_GetTime;
	bBusy				: BOOL;
	bError          	: BOOL :=FALSE;
	nErrID          	: UDINT;
	presetTime      	: TIMESTRUCT;
	syncTimer       	: TON;
	syncTrigger     	: F_TRIG;
	bSynchronize		: BOOL;
	fbRTC_EX2       	: RTC_EX2;
	nMicroseconds   	: DWORD;
	sNetId 				:STRING := '172.16.5.8.1.1';
	LokalClock: STRING(255);
END_VAR

// note: this text did not pass the execution check against the stored diagram
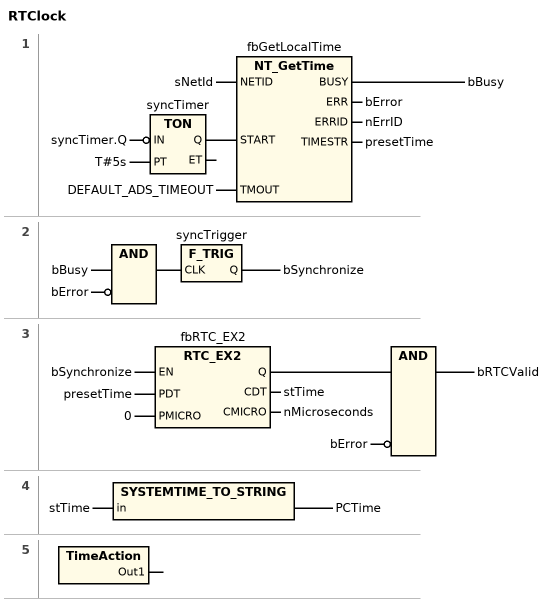
// NETWORK 1
syncTimer(IN := NOT syncTimer.Q, PT := T#5s); // TON
fbGetLocalTime(
    NETID := sNetId,
    START := syncTimer.Q,
    TMOUT := DEFAULT_ADS_TIMEOUT,
    ERR => bError,
    ERRID => nErrID,
    TIMESTR => presetTime); // NT_GetTime
bBusy := fbGetLocalTime.BUSY;

// NETWORK 2
syncTrigger(CLK := bBusy AND NOT bError); // F_TRIG
bSynchronize := syncTrigger.Q;

// NETWORK 3
fbRTC_EX2(EN := bSynchronize, PDT := presetTime, PMICRO := 0, CDT => stTime, CMICRO => nMicroseconds); // RTC_EX2
bRTCValid := fbRTC_EX2.Q AND NOT bError;

// NETWORK 4
PCTime := SYSTEMTIME_TO_STRING(in := stTime);

// NETWORK 5
TimeAction();

ACTION TimeAction:
LokalClock :=DELETE(STR:=PCTime , LEN:=4 , POS:= 20);
IF stTime.wMonth = OldMounth THEN
ChangeOfMounth:= FALSE ;
ELSE
ChangeOfMounth:= TRUE ;
END_IF
IF stTime.wHour = OldHour THEN
bHourChanged := FALSE;
ELSE
bHourChanged:= TRUE;
END_IF
IF stTime.wDay = OldDay THEN
ChangeOfDay := FALSE;
ELSE
ChangeOfDay:= TRUE;
END_IF
IF stTime.wMinute = OldMinute THEN
bMinuteChanged := FALSE ;
ELSE
bMinuteChanged:= TRUE;
END_IF
IF stTime.wHour >17 OR stTime.wHour  <8 THEN
WorkingHour := FALSE;
ELSE
WorkingHour:=TRUE;
END_IF
IF stTime.wDayOfWeek > 0 THEN
ChangeOfweek := TRUE;
ELSE
ChangeOfweek:= FALSE;
END_IF
IF stTime.wDayOfWeek = 0 OR  stTime.wDayOfWeek =  6 THEN
bWeekend := TRUE;
ELSE
bWeekend:= FALSE;
END_IF
END_ACTION

END_PROGRAM

// ---- GlobalTextList.TcGTLO
TEXTLIST GlobalTextList
  427 = '%s'
  29 = 'Air\nBedrom'
  28 = 'Air\nBjorn'
  677 = 'Bedroom'
  491 = 'Bedroom %2.1f'
  411 = 'Bjorn'
  886 = 'Bjorn %2.1f'
  956 = 'Closett'
  517 = 'Office %2.1f'
  731 = 'Ofice %2.1f'
  62 = 'PT100_Bathroom %2.1f'
  475 = 'PT100_CX1000 %2.1f'
  241 = 'PT100_Outside %2.1f'
  265 = 'Spotlight'
  33 = 'Stairlight'
  204 = 'Toilet'
  123 = 'TotalCurrent %2.1f'
  109 = 'Wew Room'
END_TEXTLIST

// ---- VISUs/VisuEnocean/TC_VISU.TcVIS
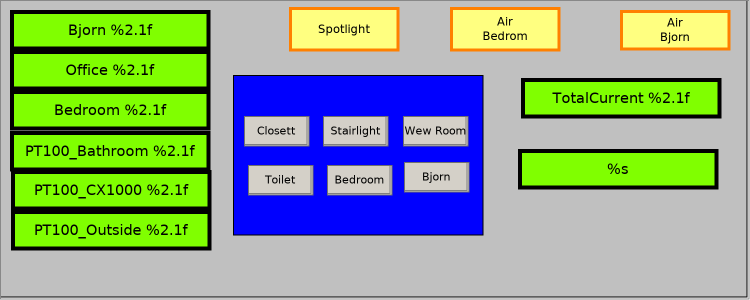
VISUALIZATION TC_VISU  // 750x300
    Rectangle (-3,-3 750x300), text variable: .PCTime
    RoundedRectangle (10,10 200x40), "Bjorn %2.1f", text variable: INT_TO_REAL(.BjornTemp )/10
    RoundedRectangle (10,50 200x40), "Office %2.1f", text variable: INT_TO_REAL (.OfficeTemp) /10
    RoundedRectangle (10,90 200x40), "Bedroom %2.1f", text variable: INT_TO_REAL (.BedRoomTemp) /10
    RoundedRectangle (521,78 200x40), "TotalCurrent %2.1f", text variable: INT_TO_REAL(.TotalCurrent )/10
    RoundedRectangle (620,10 110x40), "Air Bjorn", text variable: AirBjorn, colour toggle: AirBjorn
        toggle AirBjorn
    RoundedRectangle (450,7 110x44), "Air Bedrom", text variable: AirBedroom, colour toggle: AirBedroom
        toggle AirBedroom
    RoundedRectangle (233,75 250x160)
    Button (244,116 65x30), "Closett", text variable: WalkingClosett, colour toggle: WalkingClosett
        toggle WalkingClosett
    Button (323,116 65x30), "Stairlight", text variable: StairLight, colour toggle: StairLight
        toggle StairLight
    Button (403,116 65x30), "Wew Room", colour toggle: Livingroom
        toggle Livingroom p2164770859=TRUE
    Button (248,165 65x30), "Toilet", text variable: ToiletLight, colour toggle: ToiletLight
        toggle ToiletLight
    Button (327,165 65x30), "Bedroom", text variable: BedRoomLight, colour toggle: BedRoomLight
        toggle BedRoomLight
    Button (404,162 65x30), "Bjorn", text variable: BjornLight, colour toggle: BjornLight
        toggle BjornLight
    RoundedRectangle (289,7 110x44), "Spotlight", text variable: SpotLight, colour toggle: SpotLight
        toggle SpotLight
    RoundedRectangle (10,131 200x40), "PT100_Bathroom %2.1f", text variable: INT_TO_REAL(.PT100_Bathroom)/10
        p4168582468: TotalCurrent )/10
    RoundedRectangle (11,170 200x40), "PT100_CX1000 %2.1f", text variable: INT_TO_REAL(PT100_CX1000 )/10
        p4168582468: INT_TO_REAL(.TotalCurrent )/10
    RoundedRectangle (11,210 200x40), "PT100_Outside %2.1f", text variable: INT_TO_REAL(PT100_Outside)/10
    RoundedRectangle (518,149 200x40), "%s", text variable: .RTClock .LokalClock
END_VISUALIZATION
